// TIA Portal project "DENEME_2022_06_23" (V16)

(* hardware
DEVICE "S71500/ET200MP station_1"  S7-1500 station
   slot 0: "Rail_0"  Rack  6ES7 590-1***0-0AA0
   slot 1: "PLC_1"  CPU 1511C-1 PN  6ES7 511-1CK01-0AB0  V2.8
      slot 3: "CPU display_1"  6ES7591-1AA00-0AA0
      slot 32768: "PROFINET interface_1"  X1
         slot 32769: "Port_1"  X1 P1
         slot 32770: "Port_2"  X1 P2
      slot 34817: "Virtual CP interface port_1"  Virtual CP interface port  Virtual CP interface port
*)

// ===== PLC "PLC_1"  CPU 1511C-1 PN =====

VAR_GLOBAL   // PLC tag table "Default tag table"
   "START" AT %I0.0 : Bool;
   "STOP" AT %I0.1 : Bool;
   "L1" AT %I0.2 : Bool;
   "L2" AT %I0.3 : Bool;
   "H2" AT %I0.4 : Bool;
   "MOTOR" AT %Q0.0 : Bool;
   "MOTOR_MEM" AT %M5.0 : Bool;
END_VAR

FUNCTION "POOL&TANK EXAMPLE" : Void   // FC1, LAD
{ S7_Optimized_Access := 'TRUE' }
VERSION : 0.1
BEGIN

REGION Network 1
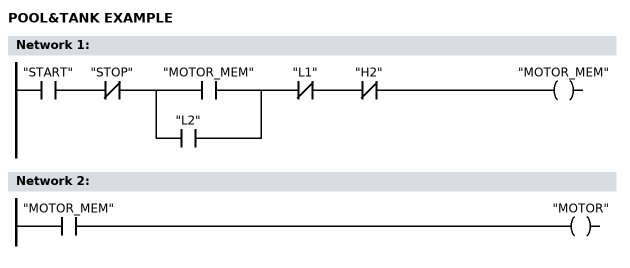
   RUNG wire#powerrail
      Contact( "START" )
      I_Contact( "STOP" )
      wire#w1
      Contact( "MOTOR_MEM" )
      wire#w2
      I_Contact( "L1" )
      I_Contact( "H2" )
      Coil( "MOTOR_MEM" )
   END_RUNG
   RUNG wire#w1
      Contact( "L2" )
   END_RUNG wire#w2
   // the same network as SCL:
   "MOTOR_MEM" := "START" AND NOT "STOP" AND ("MOTOR_MEM" OR "L2") AND NOT "L1" AND NOT "H2";
END_REGION

REGION Network 2
   RUNG wire#powerrail
      Contact( "MOTOR_MEM" )
      Coil( "MOTOR" )
   END_RUNG
   // the same network as SCL:
   "MOTOR" := "MOTOR_MEM";
END_REGION
END_FUNCTION

ORGANIZATION_BLOCK "Main"   // OB1, LAD, ProgramCycle
TITLE = "Main Program Sweep (Cycle)"
{ S7_Optimized_Access := 'TRUE' }
VERSION : 0.1
   VAR_INPUT
      Initial_Call : Bool;   // Initial call of this OB
      Remanence : Bool;   // =True, if remanent data are available
   END_VAR
BEGIN

REGION Network 1
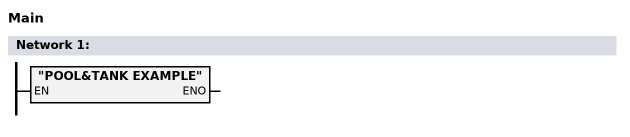
   RUNG wire#powerrail
      "POOL&TANK EXAMPLE"()
   END_RUNG
   // the same network as SCL:
   "POOL&TANK EXAMPLE"();
END_REGION
END_ORGANIZATION_BLOCK